// TwinCAT 3 PLC project SystemEngineering_PLC
// ProgramVersion: 3.1.4026.11
// libraries:
//   Tc2_Standard, * (Beckhoff Automation GmbH)
//   Tc2_System, * (Beckhoff Automation GmbH)
//   Tc3_EventLogger, * (Beckhoff Automation GmbH)
//   Tc3_JsonXml, * (Beckhoff Automation GmbH)
// project tree:
//   DUTs/ ST_HmiEventJson.TcDUT
//   / PlcTask.TcTTO
//   POUs/02_Projecttools/Actuator/ FB_Cylinder.TcPOU, ST_CylinderConfig.TcDUT
//   POUs/02_Projecttools/Sensors/ FB_Input.TcPOU
//   POUs/10_Machine/01_InfeedContainer/ FB_InfeedContainerUnit.TcPOU
//   POUs/10_Machine/02_InfeedFood/ FB_InfeedFoodUnit.TcPOU
//   POUs/10_Machine/03_Inspection/ FB_InspectionUnit.TcPOU
//   POUs/10_Machine/04_Labeling/ FB_LabelingUnit.TcPOU
//   POUs/10_Machine/05_Sealing/ FB_SealingUnit.TcPOU
//   POUs/10_Machine/06_Outfeed/ FB_OutfeedUnit.TcPOU
//   POUs/10_Machine/ FB_BaseMainStation.TcPOU, FB_MachineUnit.TcPOU
//   POUs/ MAIN.TcPOU
// real-time tasks:
//   TASK PlcTask: cycle T#10ms, priority 20, ADS port 350

CONFIGURATION SystemEngineering_PLC
    RESOURCE PLC ON TwinCAT3
        TASK PlcTask(INTERVAL := T#10ms, PRIORITY := 20);
        PROGRAM MAIN WITH PlcTask : MAIN;
    END_RESOURCE
END_CONFIGURATION

// ---- DUTs/ST_HmiEventJson.TcDUT
TYPE ST_HmiEventJson :
STRUCT
	eplan				: STRING;
	popUp				: BOOL;
END_STRUCT
END_TYPE

// ---- POUs/02_Projecttools/Actuator/ST_CylinderConfig.TcDUT
TYPE ST_CylinderConfig :
STRUCT
	{attribute 'TcHmiSystemEng.Parameter.Name' := 'Disable Feedback'}
	{attribute 'TcHmiSystemEng.Parameter.Info' := 'Disable the feedback for the base position'}
	{attribute 'TcHmiSystemEng.Parameter.GroupName' := 'Base Position'} 
	{attribute 'TcHmiSystemEng.Parameter.Layer' := '-1'}
	_disableFeedbackBP		: BOOL;
	{attribute 'TcHmiSystemEng.Parameter.Name' := 'Disable Feedback'}
	{attribute 'TcHmiSystemEng.Parameter.Info' := 'Disable the feedback for the work position'}
	{attribute 'TcHmiSystemEng.Parameter.GroupName' := 'Work Position'} 
	{attribute 'TcHmiSystemEng.Parameter.Layer' := '-1'}
	_disableFeedbackWP		: BOOL;
	{attribute 'TcHmiSystemEng.Parameter.Name' := 'Invert Feedback'}
	{attribute 'TcHmiSystemEng.Parameter.Info' := 'Invert the feedback for the work position'}
	{attribute 'TcHmiSystemEng.Parameter.GroupName' := 'Base Position'} 
	{attribute 'TcHmiSystemEng.Parameter.Layer' := '-1'}
	_invertFeedbackBP		: BOOL;
	{attribute 'TcHmiSystemEng.Parameter.Name' := 'Invert Feedback'}
	{attribute 'TcHmiSystemEng.Parameter.Info' := 'Invert the feedback for the work position'}
	{attribute 'TcHmiSystemEng.Parameter.GroupName' := 'Work Position'} 
	{attribute 'TcHmiSystemEng.Parameter.Layer' := '-1'}
	_invertFeedbackWP		: BOOL;
	
	{attribute 'TcHmiSystemEng.Parameter.Name' := 'Timeout'}
	{attribute 'TcHmiSystemEng.Parameter.Info' := 'Work process timout'}
	{attribute 'TcHmiSystemEng.Parameter.Min' := 'T#0S'}
	{attribute 'TcHmiSystemEng.Parameter.Max' := 'T#30S'}
	{attribute 'TcHmiSystemEng.Parameter.GroupName' := 'Time'}
	{attribute 'TcHmiSystemEng.Parameter.Layer' := '-1'}
	_timeout 				: TIME := T#5S;
	
	{attribute 'TcHmiSystemEng.Parameter.Name' := 'Simulation Feedback'}
	{attribute 'TcHmiSystemEng.Parameter.Info' := 'Work process simulation time'}
	{attribute 'TcHmiSystemEng.Parameter.Min' := 'T#0S'}
	{attribute 'TcHmiSystemEng.Parameter.Max' := 'T#30S'}
	{attribute 'TcHmiSystemEng.Parameter.GroupName' := 'Time'}
	{attribute 'TcHmiSystemEng.Parameter.Layer' := '-1'}
	_simulationFeedback		: TIME	:= T#3S;
END_STRUCT
END_TYPE

// ---- POUs/MAIN.TcPOU
PROGRAM MAIN
VAR
	{attribute 'TcHmiSystemEng.Parameter.Name' 				:= 'Machine'}
	{attribute 'TcHmiSystemEng.Parameter.TreeViewImage'	 	:= 'Portal/normal.svg'}	
	fbMachine					: FB_MachineUnit;
	
	_isInit      				: BOOL;
END_VAR

END_PROGRAM

// ---- POUs/10_Machine/FB_MachineUnit.TcPOU
FUNCTION_BLOCK FB_MachineUnit
VAR	
	{attribute 'TcHmiSystemEng.Parameter.Name' := 'Machine name'}
	{attribute 'TcHmiSystemEng.Parameter.Info' := 'Enter the name from the machine'}
	_sMachineName				: STRING;
	{attribute 'TcHmiSystemEng.Parameter.Name' := 'Machine version'}
	{attribute 'TcHmiSystemEng.Parameter.Info' := 'Enter the version from the machine'}
	_sMachineVersion			: STRING := '1.0.0.0';
		
	// stations
	{attribute 'TcHmiSystemEng.Parameter.Name' 				:= 'Infeed Container'}
	{attribute 'TcHmiSystemEng.Parameter.TreeViewImage'	 	:= 'Conveyor/normal.svg'}	
	_fbInfeedContainer			: FB_InfeedContainerUnit;
	{attribute 'TcHmiSystemEng.Parameter.Name' 				:= 'Infeed Food'}
	{attribute 'TcHmiSystemEng.Parameter.TreeViewImage'	 	:= 'TrayFeeder/normal.svg'}	
	_fbInfeedFood				: FB_InfeedFoodUnit;
	{attribute 'TcHmiSystemEng.Parameter.Name' 				:= '@this._sStationName'}
	{attribute 'TcHmiSystemEng.Parameter.TreeViewImage'	 	:= '@this._sImage'}	
	_fbInspection				: FB_InspectionUnit;
	{attribute 'TcHmiSystemEng.Parameter.Name' 				:= 'Labeling'}
	{attribute 'TcHmiSystemEng.Parameter.TreeViewImage'	 	:= 'Packaging/normal.svg'}	
	_fbLabeling					: FB_LabelingUnit;
	{attribute 'TcHmiSystemEng.Parameter.Name' 				:= 'Sealing'}
	{attribute 'TcHmiSystemEng.Parameter.TreeViewImage'	 	:= 'Temperature/normal.svg'}
	_fbSealing					: FB_SealingUnit;
	{attribute 'TcHmiSystemEng.Parameter.Name' 				:= 'Outfeed'}
	{attribute 'TcHmiSystemEng.Parameter.TreeViewImage'	 	:= 'Handling/normal.svg'}	
	_fbOutfeed					: FB_OutfeedUnit;
END_VAR


// cycle
Ac_Cycle();

ACTION Ac_Cycle:

_fbInfeedContainer();
_fbInfeedFood();
_fbInspection();
_fbLabeling();
_fbSealing();
_fbOutfeed();
END_ACTION

END_FUNCTION_BLOCK

// ---- POUs/10_Machine/01_InfeedContainer/FB_InfeedContainerUnit.TcPOU
FUNCTION_BLOCK FB_InfeedContainerUnit EXTENDS FB_BaseMainStation
VAR CONSTANT
END_VAR
VAR_INPUT
END_VAR
VAR_OUTPUT
END_VAR
VAR	
	{ attribute 'TcHmiSystemEng.Parameter.Name' := 'Cut Cylinder' }
	_fbCutCylinder			: FB_Cylinder;
	{ attribute 'TcHmiSystemEng.Parameter.Name' := 'Press Cylinder' }
	_fbPressCylinder		: FB_Cylinder;
END_VAR

END_FUNCTION_BLOCK

// ---- POUs/10_Machine/FB_BaseMainStation.TcPOU
FUNCTION_BLOCK FB_BaseMainStation
VAR_INPUT
END_VAR
VAR_OUTPUT
END_VAR
VAR
	{attribute 'TcHmiSystemEng.Parameter.Name' := 'Station name'}
	{attribute 'TcHmiSystemEng.Parameter.Info' := 'Enter the name from the station'}
	_sStationName					: STRING;
END_VAR

END_FUNCTION_BLOCK

// ---- POUs/02_Projecttools/Actuator/FB_Cylinder.TcPOU
{attribute 'TcHmiSystemEng.Parameter.TreeViewImage'	 	:= 'Cylinder/normal.svg'}
FUNCTION_BLOCK FB_Cylinder
VAR_OUTPUT CONSTANT	
END_VAR
VAR_INPUT
	quit									: BOOL;	//Resets error with rising edge
	toWorkPos								: BOOL;	//moves cylinder to work position
	toBasePos								: BOOL	:= TRUE;	//moves cylinder to base position

	feedBasePos								: BOOL := TRUE;	//enables feed in base direction
	feedWorkPos								: BOOL := TRUE;	//enables feed in work direction
	
	hmiEventDataAlarmErrBasePos				: ST_HmiEventJson;
	hmiEventDataAlarmErrWorkPos				: ST_HmiEventJson;
END_VAR                                     			
VAR_OUTPUT       			
	inBasePos								: BOOL;	//TRUE when cylinder is in base position
	inWorkpos								: BOOL;	//TRUE when cylinder is in work position
	done									: BOOL; //Limit sensor reached or feedback time counted down
	busy									: BOOL;	//Busy is TRUE at the rising edge of Execute and FALSE when one of the outputs Done, Aborted, or Error is set 
	errBasePos								: BOOL;	//Cannot reach base position
	errWorkPos								: BOOL;	//Cannot reach work position  
	errLogic								: BOOL; 	//Both Feedbacks signaled

	q_ToBasePos						AT  %Q* : BOOL; //Hardware output
	q_ToWorkPos						AT  %Q* : BOOL; //Hardware output
END_VAR
VAR	
	{attribute 'TcHmiSystemEng.Parameter.Name' := 'Name'}
	{attribute 'TcHmiSystemEng.Parameter.Info' := 'Name of the cylinder'}
	_name									: STRING;
	{attribute 'TcHmiSystemEng.Parameter.Name' := 'Id'}
	{attribute 'TcHmiSystemEng.Parameter.Info' := 'Identification name of the cylinder'}
	_id										: STRING;
	
	_sensorBasePos							: FB_Input;
	_sensorWorkPos							: FB_Input;
	_ton_ErrWorkPos							: TON;
	_ton_ErrBasePos							: TON;
	
	{ attribute 'TcHmiSystemEng.Parameter.Name' := 'Config' }
	_config									: ST_CylinderConfig;
	
	_alarmErrBasePos						: FB_TcAlarm;	
	_alarmErrWorkPos						: FB_TcAlarm;
	_alarmErrLogic							: FB_TcAlarm;
	
  	_fbJsonDataType							: FB_JsonReadWriteDataType;
  	_sJsonDoc      							: STRING(2000); 
END_VAR

	(* Cylinder	 IO V2.8					 								       	*)
	(* Includes functionblock "INPUT" 												*)
	(********************************************************************************)

(* Messages *********************************************************)
	Messages();
	
(* Write Output *****************************************************)
		
	IF toBasePos AND toWorkPos 
	THEN
		ON();
	ELSIF toBasePos 	
	THEN
		BasePos();
	ELSIF toWorkPos 
	THEN
		WorkPos();
	ELSE
		OFF();
	END_IF

(* Reedkontakte lesen ***********************************************)
	_sensorBasePos(
		force	:= q_ToBasePos AND NOT inWorkpos AND _config._disableFeedbackBP,
		invert	:= _config._invertFeedbackBP,
		pt_ON	:= SEL(_config._disableFeedbackBP ,T#0MS,_config._simulationFeedback),
		pt_OFF	:= ,
		q_DIRECT=>,
		q		=> inBasePos,
		q_RT	=> ,
		q_FT	=> ,
		in		=> );

	_sensorWorkPos(
		force	:= q_ToWorkPos AND NOT inBasePos AND _config._disableFeedbackWP,
		invert	:= _config._invertFeedbackWP,
		pt_ON	:= SEL(_config._disableFeedbackWP ,T#0MS,_config._simulationFeedback),
		pt_OFF	:= ,
		q_DIRECT=>,
		q		=> inWorkpos,
		q_RT	=> ,
		q_FT	=> ,
		in		=> );
                        	
(* ack Error **********************************************************)
	IF quit  THEN  Quitting(); END_IF

(* Timeout WorkPos ************************************************)
	_ton_ErrWorkPos(	IN := q_ToWorkPos AND (NOT inWorkpos OR inBasePos),
					PT := MAX(_config._timeout,_config._simulationFeedback + T#1S),
					Q => errWorkPos);

(* Timeout WorkPos ************************************************)
	_ton_ErrBasePos(	IN := q_ToBasePos AND (NOT inBasePos OR inWorkpos),
					PT := MAX(_config._timeout,_config._simulationFeedback + T#1S),
					Q => errBasePos);

(* Senor logic ******************************************************)
	errLogic								:= inBasePos AND inWorkpos;
	
(*********************************************************************)

METHOD PUBLIC BasePos : BOOL //Return = Done -> InBasePos
toWorkPos 				:= q_ToWorkPos		:= FALSE;
toBasePos 									:= TRUE;
q_ToBasePos	 								:= feedBasePos AND NOT inBasePos;
BasePos 				:= done				:= inBasePos;
busy										:= NOT done;
END_METHOD

METHOD PUBLIC Enable : BOOL //Return Done = TRUE if WorkPos is TRUE and InWorkPos = TRUE or WorkPos is FALSE and InBasePos is TRUE 
VAR_INPUT
	workPos													:	BOOL;
END_VAR
IF workPos
THEN
	Enable 									:= THIS^.workPos();
ELSE
	Enable 									:= THIS^.basePos();
END_IF
END_METHOD

PROPERTY PUBLIC InError : Bool
GET
InError := errBasePos OR errWorkPos OR errLogic;
END_GET
END_PROPERTY

{attribute 'call_after_global_init_slot' := '100'}
METHOD Init : BOOL
VAR_INPUT
END_VAR

_alarmErrBasePos.CreateEx(TC_EVENTS.Cylinder.errBasePos, FALSE, 0);
_alarmErrBasePos.ipArguments.AddString(_id);

_alarmErrWorkPos.CreateEx(TC_EVENTS.Cylinder.errWorkPos, FALSE, 0);
_alarmErrWorkPos.ipArguments.AddString(_id);

_alarmErrLogic.CreateEx(TC_EVENTS.Cylinder.errLogic, FALSE, 0);
_alarmErrLogic.ipArguments.AddString(_id);
END_METHOD

ACTION Messages:

// errBasePos
IF errBasePos THEN
	// JSON
	_sJsonDoc := _fbJsonDataType.GetJsonStringFromSymbol('ST_HmiEventJson', SIZEOF(hmiEventDataAlarmErrBasePos), ADR(hmiEventDataAlarmErrBasePos));
	_alarmErrBasePos.SetJsonAttribute(_sJsonDoc);
	_alarmErrBasePos.Raise(0);
ELSE
	_alarmErrBasePos.Clear(0, TRUE);
END_IF
// errWorkPos
IF errWorkPos THEN	
	// JSON
	_sJsonDoc := _fbJsonDataType.GetJsonStringFromSymbol('ST_HmiEventJson', SIZEOF(hmiEventDataAlarmErrWorkPos), ADR(hmiEventDataAlarmErrWorkPos));
	_alarmErrWorkPos.SetJsonAttribute(_sJsonDoc);
	_alarmErrWorkPos.Raise(0);
ELSE	
	_alarmErrWorkPos.Clear(0, TRUE);
END_IF
// errLogic
IF errLogic THEN	
	_alarmErrLogic.Raise(0);
ELSE
	_alarmErrLogic.Clear(0, TRUE);
END_IF
END_ACTION

PROPERTY PUBLIC NoFeed : BOOL
GET
NoFeed := toWorkPos and not feedWorkPos or toBasePos and not feedBasePos;
END_GET
END_PROPERTY

METHOD PUBLIC Off : BOOL //Result = Done
done := busy := q_ToWorkPos := q_ToBasePos 		:= FALSE;
toBasePos := toWorkPos 							:= FALSE;
Off												:= TRUE;
END_METHOD

METHOD PUBLIC On : BOOL //Result = Done
toWorkPos 					:= q_ToWorkPos 	:= feedWorkPos;
toBasePos 					:= q_ToBasePos	:= feedBasePos;
done 										:= TRUE;
busy 										:= TRUE;
On											:= TRUE;
END_METHOD

METHOD PUBLIC Quitting : BOOL //Result = Quitting active
_ton_ErrWorkPos(IN := FALSE);
_ton_ErrBasePos(IN := FALSE);
errWorkPos	:= errBasePos := errLogic		:= FALSE;
Quitting									:= FALSE;
END_METHOD

METHOD PUBLIC WorkPos : BOOL //Return = Done -> InWorkPos
toBasePos 				:= q_ToBasePos 		:= FALSE;
toWorkPos									:= TRUE;
q_ToWorkPos	 								:= feedWorkPos AND NOT inWorkpos;
WorkPos					:= done 			:= inWorkpos;
Busy										:= NOT done;
END_METHOD

END_FUNCTION_BLOCK

// ---- POUs/02_Projecttools/Sensors/FB_Input.TcPOU
FUNCTION_BLOCK FB_Input
VAR_INPUT
	force													:	BOOL := FALSE; 	//simulates Input
	invert													:	BOOL := FALSE; 	//inverts the Hardware Input
	pt_ON													:	TIME := T#0MS;	//on delay
	pt_OFF													:	TIME := T#0MS;	//off delay
END_VAR             										
VAR_OUTPUT          										
	q														:	BOOL;	//Signal Delay
	q_RT													:	BOOL;	//R_Trig Signal of Q
	q_FT													:	BOOL;	//F_Trig Signal of Q
	q_DIRECT												:	BOOL; 	//Signal direct
	in												AT  %I* : 	BOOL; 	//Hardware Input
END_VAR
VAR
	ton														:	TON;
END_VAR

(* Input/Sensor Functionblock with On/Off	attenuation and rising / fallen edge 	V2.0	*)
(********************************************************************************************)

(************************************)
IF NOT q THEN
	ton(IN := (in OR force) XOR invert, PT := pt_ON);
	q 														:= ton.Q;
	q_RT 													:= q;
	q_FT 													:= FALSE;
	q_DIRECT 												:= ton.IN;
ELSE
	ton(IN := NOT ((in OR force) XOR invert), PT := pt_OFF);
	q 														:= q AND NOT ton.Q;
	q_RT 													:= FALSE;
	q_FT 													:= NOT q;
	q_DIRECT 												:= q AND NOT ton.IN;
END_IF
(********************************************************************************************)

END_FUNCTION_BLOCK

// ---- POUs/10_Machine/02_InfeedFood/FB_InfeedFoodUnit.TcPOU
FUNCTION_BLOCK FB_InfeedFoodUnit EXTENDS FB_BaseMainStation
VAR_INPUT
END_VAR
VAR_OUTPUT
END_VAR
VAR	
	{ attribute 'TcHmiSystemEng.Parameter.Name' := 'Cut Cylinder' }
	_fbCutCylinder			: FB_Cylinder;
END_VAR

END_FUNCTION_BLOCK

// ---- POUs/10_Machine/03_Inspection/FB_InspectionUnit.TcPOU
FUNCTION_BLOCK FB_InspectionUnit EXTENDS FB_BaseMainStation
VAR CONSTANT
END_VAR
VAR_INPUT
END_VAR
VAR_OUTPUT
END_VAR
VAR
	{attribute 'TcHmiSystemEng.Parameter.Name' := 'Station Image'}
	{attribute 'TcHmiSystemEng.Parameter.Info' := 'Image of the station'}
	_sImage					: STRING := 'Vision/normal.svg';
	{attribute 'TcHmiSystemEng.Parameter.Name' := 'Resolution'}
	{attribute 'TcHmiSystemEng.Parameter.Info' := 'Resolution of the image'}
    {attribute 'TcHmiSystemEng.Parameter.Unit' := 'TcHmiSystemEng.Preset.Unit'}
    {attribute 'TcHmiSystemEng.Parameter.Min' := '@_nMinResolution'}
    {attribute 'TcHmiSystemEng.Parameter.Max' := '@_nMaxResolution'}
    _nResolution			: REAL;
    _nMinResolution			: REAL := 30;
    _nMaxResolution			: REAL := 100;
END_VAR

END_FUNCTION_BLOCK

// ---- POUs/10_Machine/04_Labeling/FB_LabelingUnit.TcPOU
FUNCTION_BLOCK FB_LabelingUnit EXTENDS FB_BaseMainStation
VAR_INPUT
END_VAR
VAR_OUTPUT
END_VAR
VAR 
	{attribute 'TcHmiSystemEng.Parameter.Name' := 'Label Speed'}
	{attribute 'TcHmiSystemEng.Parameter.Info' := 'Enter the speed of the label'}
    {attribute 'TcHmiSystemEng.Parameter.Unit' := 'mm/1'}
    {attribute 'TcHmiSystemEng.Parameter.Min' := '@_nMinSpeed'}
    {attribute 'TcHmiSystemEng.Parameter.Max' := '@_nMaxSpeed'}
    _nSpeed        : REAL;
    _nMinSpeed     : REAL := 0;
    _nMaxSpeed     : REAL := 3000;
END_VAR

END_FUNCTION_BLOCK

// ---- POUs/10_Machine/05_Sealing/FB_SealingUnit.TcPOU
FUNCTION_BLOCK FB_SealingUnit EXTENDS FB_BaseMainStation
VAR_INPUT
END_VAR
VAR_OUTPUT
END_VAR
VAR
	{attribute 'TcHmiSystemEng.Parameter.Name' := 'Temperature'}
	{attribute 'TcHmiSystemEng.Parameter.Info' := 'Temperature of the sealing'}
    {attribute 'TcHmiSystemEng.Parameter.Unit' := '°C'}
    {attribute 'TcHmiSystemEng.Parameter.Min' := '@_nMinTemperature'}
    {attribute 'TcHmiSystemEng.Parameter.Max' := '@_nMaxTemperature'}
    _nTemperature        : REAL;
    _nMinTemperature     : REAL := 30;
    _nMaxTemperature     : REAL := 100;
END_VAR

END_FUNCTION_BLOCK

// ---- POUs/10_Machine/06_Outfeed/FB_OutfeedUnit.TcPOU
FUNCTION_BLOCK FB_OutfeedUnit EXTENDS FB_BaseMainStation
VAR_INPUT
END_VAR
VAR_OUTPUT
END_VAR
VAR
	{attribute 'TcHmiSystemEng.Parameter.Name' := 'Label Speed'}
	{attribute 'TcHmiSystemEng.Parameter.Info' := 'Enter the speed of the label'}
    {attribute 'TcHmiSystemEng.Parameter.Unit' := 'mm/1'}
    {attribute 'TcHmiSystemEng.Parameter.Min' := '0'}
    {attribute 'TcHmiSystemEng.Parameter.Max' := '@_nMaxPickPosition'}
    _nPickPosition        : REAL;
    _nMaxPickPosition     : REAL := 3000;
END_VAR

END_FUNCTION_BLOCK
